{attribute 'GeneratedUsingTerminal: EL2642-0000-0016'}
{attribute addProperty BoxType "EL2642-0000-0016"}
{attribute addProperty Id "Outputs_Group_2AT %Q*Outputs_Group_78994C084"}
{attribute addProperty CRC "2189460104"}
{attribute addProperty Size "4"}
TYPE DO_Group_2_Outputs_82808288 :
STRUCT
	{attribute addProperty Name "Outputs_Group_2"}
	Outputs_Group_2 AT %Q* : Outputs_Group_78994C08;
END_STRUCT
END_TYPE

(* stored: Version 1.2.0.0, ProductVersion 3.1.4024.9
   DUT DO_Group_2_Outputs_82808288: Id {9a59dd3a-4361-4eda-8554-bafb70ed9e31} *)
